(* CODESYS project proSlotStruct.export

Project tree, tasks and I/O mapping:
  data type ST_WarehouseSlot
*)

// ST_WarehouseSlot
TYPE ST_WarehouseSlot :
STRUCT
    iCurrentCount : INT := 0;      // How many items are inside
    iMaxCapacity  : INT := 1;      // How many it CAN hold (1, 2, 3...)
    sDisplayText  : STRING := '';  // Will show "2 / 5"
    dwColor       : DWORD := 16#FF00FF00; // Default Green (ARGB format)
	sItemName: STRING(255);
END_STRUCT
END_TYPE
